// TIA Portal V17 export
// export: Created 2024-01-30T08:49:17.224959Z, ExportSetting WithDefaults, DisplayName Totally Integrated Automation Portal, DisplayVersion V17 Update 6, DisplayName TIA Portal Openness, DisplayVersion V17 Update 6, DisplayName TIA Portal Version Control Interface, DisplayVersion V17, DisplayName STEP 7 Professional, DisplayVersion V17 Update 6, DisplayName STEP 7 Safety, DisplayVersion V17 Update 6, DisplayName WinCC Advanced, DisplayVersion V17 Update 6
TYPE "UDT_ProGloveScanDat"
// stored: IsFailsafeCompliant false
   STRUCT
      Location_ID : DInt;
      Tray_ID : UInt;
      Tray_ScanTime : Date_And_Time;
      Zelle_ID : UInt;
      Zelle_ScanTime : Date_And_Time;
   END_STRUCT;
END_TYPE
